FUNCTION SPLIT_BYTE_INTO_BOOLS (* this Function extracts the 8 BOOLS from a byte *)
  (* Standard: 61499-1; Description: Copyright (c) 2024 HR Agrartechnik GmbH This program and the accompanying materials are made available under the terms of the Eclipse Public License 2.0 which is available at https://www.eclipse.org/legal/epl-2.0/ SPDX-License-Identifier: EPL-2.0 *)
  (* Version 3.0, 2025-04-14, Patrick Aigner, changed package *)
  (* Version 1.1, 2024-07-28, Moritz Ortmeier, HR Agrartechnik, rename Function and change Output Variables *)
  (* Version 1.0, 2024-02-22, Franz Höpfinger, HR Agrartechnik, initial Implementation *)
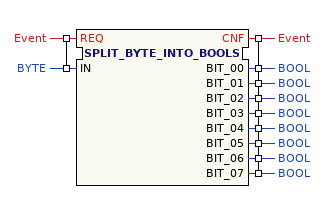
  EVENT_INPUT
    REQ WITH IN;
  END_EVENT
  EVENT_OUTPUT
    CNF WITH BIT_00, BIT_01, BIT_02, BIT_03, BIT_04, BIT_05, BIT_06, BIT_07;
  END_EVENT
  VAR_INPUT
    IN : BYTE;
  END_VAR
  VAR_OUTPUT
    BIT_00 : BOOL;
    BIT_01 : BOOL;
    BIT_02 : BOOL;
    BIT_03 : BOOL;
    BIT_04 : BOOL;
    BIT_05 : BOOL;
    BIT_06 : BOOL;
    BIT_07 : BOOL;
  END_VAR
  BODY IN ST:
(* this Function extracts the 8 BOOLS from a byte *)
FUNCTION SPLIT_BYTE_INTO_BOOLS

VAR_INPUT
	IN : BYTE;
END_VAR

VAR_OUTPUT
	BIT_00 : BOOL;
	BIT_01 : BOOL;
	BIT_02 : BOOL;
	BIT_03 : BOOL;
	BIT_04 : BOOL;
	BIT_05 : BOOL;
	BIT_06 : BOOL;
	BIT_07 : BOOL;
END_VAR

BIT_00 := IN.%X0;
BIT_01 := IN.%X1;
BIT_02 := IN.%X2;
BIT_03 := IN.%X3;
BIT_04 := IN.%X4;
BIT_05 := IN.%X5;
BIT_06 := IN.%X6;
BIT_07 := IN.%X7;

END_FUNCTION
  END_BODY
END_FUNCTION
